// TwinCAT 3 PLC project PLC
// ProgramVersion: 3.1.4024.0
// libraries:
//   Tc2_Standard, * (Beckhoff Automation GmbH)
//   Tc2_System, * (Beckhoff Automation GmbH)
//   Tc3_Module, * (Beckhoff Automation GmbH)
// project tree:
//   DUTs/ DUT.TcDUT
//   / GlobalTextList.TcGTLO, PlcTask.TcTTO, Visualization Manager.TcVMO (not stored)
//   GVLs/ gHMI.TcGVL
//   POUs/FBs/ FB_Actuator.TcPOU, FB_StartingAlarm.TcPOU, FB_Contactor.TcPOU, FB_Debounce.TcPOU
//   POUs/Fs/ F_Scale.TcPOU
//   POUs/ MAIN.TcPOU, P_Control.TcPOU
//   VISUs/ VIS_Main.TcVIS
// real-time tasks:
//   TASK PlcTask: cycle T#10ms, priority 20, ADS port 350

CONFIGURATION PLC
    RESOURCE PLC ON TwinCAT3
        TASK PlcTask(INTERVAL := T#10ms, PRIORITY := 20);
        PROGRAM MAIN WITH PlcTask : MAIN;
    END_RESOURCE
END_CONFIGURATION

// ---- DUTs/DUT.TcDUT
TYPE DUT :
STRUCT
END_STRUCT
END_TYPE

// ---- GVLs/gHMI.TcGVL
{attribute 'qualified_only'}
VAR_GLOBAL
	Start: BOOL;
	Stop: BOOL;
	Reset: BOOL;
	Run: BOOL;
	Alarm: BOOL;
	Error: BOOL;	
END_VAR

// ---- POUs/MAIN.TcPOU
PROGRAM MAIN
VAR
END_VAR

P_Control();

END_PROGRAM

// ---- POUs/P_Control.TcPOU
PROGRAM P_Control
VAR
	fbStarter: FB_StartingAlarm;
	FB_Debounce_0: FB_Debounce;
	fbDebounce: FB_Debounce;
	fbContactor: FB_Contactor;
	simContactor: FB_Debounce;
END_VAR

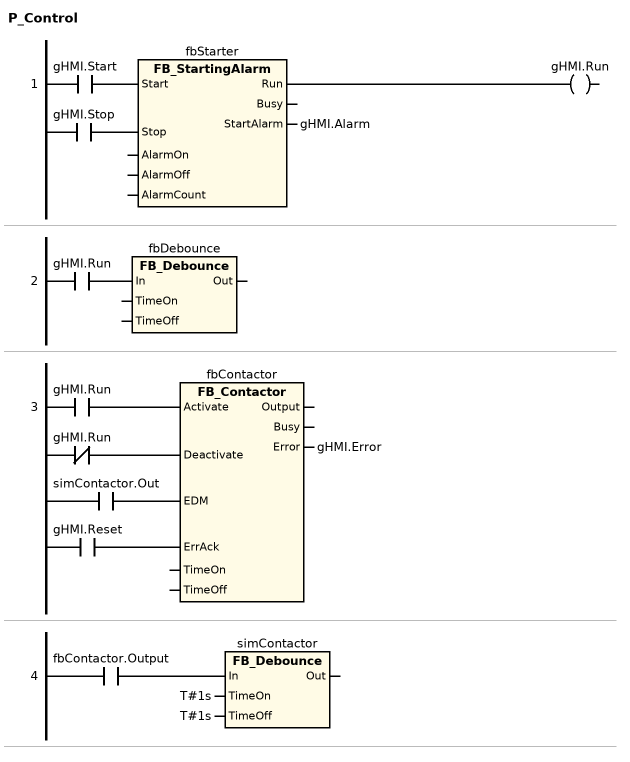
// NETWORK 1
fbStarter(Start := gHMI.Start, Stop := gHMI.Stop, StartAlarm => gHMI.Alarm); // FB_StartingAlarm
gHMI.Run := fbStarter.Run;

// NETWORK 2
fbDebounce(In := gHMI.Run); // FB_Debounce

// NETWORK 3
fbContactor(
    Activate := gHMI.Run,
    Deactivate := NOT gHMI.Run,
    EDM := simContactor.Out,
    ErrAck := gHMI.Reset,
    Error => gHMI.Error); // FB_Contactor

// NETWORK 4
simContactor(In := fbContactor.Output, TimeOn := T#1s, TimeOff := T#1s); // FB_Debounce

END_PROGRAM

// ---- POUs/FBs/FB_StartingAlarm.TcPOU
FUNCTION_BLOCK FB_StartingAlarm
VAR_INPUT
	Start: BOOL;
	Stop: BOOL;
	AlarmOn: TIME := T#500MS;
	AlarmOff: TIME := T#500MS;
	AlarmCount: UINT := 3;
END_VAR
VAR_OUTPUT
	Run: BOOL;
	Busy: BOOL;
	StartAlarm: BOOL;
END_VAR
VAR
	eState: (eInit, eIdle, eStarting, eRunning);
	eAlarmState: (eAlarmInit, eAlarmOn, eAlarmOff, eAlarmDone);
	rtrigStart: R_TRIG;
	rtrigStop: R_TRIG;
	tonAlarmOn: TON;
	tonAlarmOff: TON;
	nAlarmCount: UINT;
END_VAR

// Triggers
rtrigStop(CLK := Stop);

// Stop Interrrupt
IF rtrigStop.Q THEN
	eState := eInit;
END_IF

// State Machine
CASE eState OF
	eInit:
		Run := FALSE;
		Busy := FALSE;
		StartAlarm := FALSE;
		eAlarmState := eAlarmInit;	
		eState := eIdle;
		
	eIdle:
		IF Start THEN
			eState := eStarting;
		END_IF
		
	eStarting:
		Busy := TRUE;
		
		// Abort if Start not Held
		IF NOT Start THEN
			eState := eInit;
		END_IF
		
		// Alarm Sequence
		CASE eAlarmState OF
			eAlarmInit:
				tonAlarmOn.IN := FALSE;
				tonAlarmOn.PT := AlarmOn;
				tonAlarmOff.IN := FALSE;
				tonAlarmOff.PT := AlarmOff;
				nAlarmCount := 0;
				eAlarmState := eAlarmOn;
			eAlarmOn:
				tonAlarmOn.IN := TRUE;
				StartAlarm := TRUE;
				IF tonAlarmOn.Q THEN
					tonAlarmOn.IN := FALSE;
					eAlarmState := eAlarmOff;
				END_IF
			eAlarmOff:
				tonAlarmOff.IN := TRUE;
				StartAlarm := FALSE;
				IF tonAlarmOff.Q THEN
					tonAlarmOff.IN := FALSE;
					nAlarmCount := nAlarmCount + 1;
					IF nAlarmCount < AlarmCount THEN
						eAlarmState := eAlarmOn;
					ELSE
						eAlarmState := eAlarmDone;
					END_IF
				END_IF
				
			eAlarmDone:
				eState := eRunning;
		END_CASE
		
	eRunning:
		Busy := FALSE;
		Run := TRUE;	
END_CASE

// Call Function Blocks
tonAlarmOn();
tonAlarmOff();

END_FUNCTION_BLOCK

// ---- POUs/FBs/FB_Debounce.TcPOU
(* 	Disclaimer
	All sample code provided by Beckhoff Automation LLC are for illustrative purposes only and are provided “as is” and without any warranties, express or implied.
	Actual implementations in applications will vary significantly.
	Beckhoff Automation LLC shall have no liability for, and does not waive any rights in relation to, any code samples that it provides or the use of such code samples for any purpose.
*)
FUNCTION_BLOCK FB_Debounce
VAR_INPUT
	In: BOOL;
	TimeOn: TIME := T#2S;
	TimeOff: TIME := T#2S;
END_VAR
VAR_OUTPUT
	Out: BOOL;
END_VAR
VAR
	tonDelayOn: TON;
	tonDelayOff: TON;
END_VAR

// Set-Reset delay Timers
IF In THEN
	tonDelayOn.PT := TimeOn;
	tonDelayOn.IN := TRUE;
	tonDelayOff.IN := FALSE;
ELSE
	tonDelayOff.PT := TimeOff;
	tonDelayOff.IN := TRUE;
	tonDelayOn.IN := FALSE;
END_IF

// Set delayed Output
IF tonDelayOn.Q THEN
	Out := TRUE;
END_IF

// Reset delayed Output
IF tonDelayOff.Q THEN
	Out := FALSE;
END_IF

// Call function blocks
tonDelayOn();
tonDelayOff();

END_FUNCTION_BLOCK

// ---- POUs/FBs/FB_Contactor.TcPOU
(* 	Disclaimer
	All sample code provided by Beckhoff Automation LLC are for illustrative purposes only and are provided “as is” and without any warranties, express or implied.
	Actual implementations in applications will vary significantly.
	Beckhoff Automation LLC shall have no liability for, and does not waive any rights in relation to, any code samples that it provides or the use of such code samples for any purpose.
*)
FUNCTION_BLOCK FB_Contactor
VAR_INPUT
	Activate: BOOL;
	Deactivate: BOOL;
	EDM: BOOL;
	ErrAck: BOOL;
	TimeOn: TIME := T#3S;
	TimeOff: TIME := T#3S;
END_VAR
VAR_OUTPUT
	Output: BOOL;
	Busy: BOOL;
	Error: BOOL;
END_VAR
VAR
	eState :(eInit, eIdle, eActivate, eDeactivate, eError);
	tonWD: TON;
END_VAR

// Activating Watchdog
tonWD.IN := Output XOR EDM;
tonWD.PT := TimeOn;
IF tonWD.Q THEN
	Error := TRUE;
END_IF

// State Machine
CASE eState OF
	eInit:
		Output := FALSE;
		Busy := FALSE;
		Error := FALSE;
		eState := eIdle;
	
	eIdle:
		Busy := FALSE;
		IF Activate AND NOT Output THEN
			eState := eActivate;
		ELSIF NOT Activate AND Output THEN
			eState := eDeactivate;
		END_IF
		
	eActivate:
		Busy := TRUE;
		Output := TRUE;
		IF NOT Activate OR EDM THEN
			eState := eIdle;
		END_IF
	
	eDeactivate:
		Busy := TRUE;
		Output := FALSE;
		IF Activate OR NOT EDM THEN
			eState := eIdle;
		END_IF	
		
	eError:
		IF ErrAck THEN
			eState := eInit;
		END_IF
	
END_CASE

// Call function blocks
tonWD();

END_FUNCTION_BLOCK

// ---- POUs/FBs/FB_Actuator.TcPOU
(* 	Disclaimer
	All sample code provided by Beckhoff Automation LLC are for illustrative purposes only and are provided “as is” and without any warranties, express or implied.
	Actual implementations in applications will vary significantly.
	Beckhoff Automation LLC shall have no liability for, and does not waive any rights in relation to, any code samples that it provides or the use of such code samples for any purpose.
*)
FUNCTION_BLOCK FB_Actuator
VAR_INPUT
	Activate: BOOL;
	Deactivate: BOOL;
	EDM_Activated: BOOL;
	EDM_Deactivated: BOOL;
	ErrAck: BOOL;
	TimeOn: TIME := T#2S;
	TimeOff: TIME := T#2S;
END_VAR
VAR_OUTPUT
	Activated: BOOL;
	Busy: BOOL;
	Error: BOOL;
	ErrorId: UDINT;
END_VAR
VAR
	eState :(eInit, eIdle, eActivate, eDeactivate, eError);
	tonWD_On: TON;
	tonWD_Off: TON;
END_VAR

// Activating Watchdog
tonWD_On.IN := Activated AND NOT EDM_Activated;
tonWD_On.PT := TimeOn;
IF tonWD_On.Q THEN
	Error := TRUE;
	ErrorId := 1;
END_IF

// Deactivating Watchdog
tonWD_Off.IN := NOT Activated AND NOT EDM_Deactivated;
tonWD_Off.PT := TimeOff;
IF tonWD_Off.Q THEN
	Error := TRUE;
	ErrorId := 2;
END_IF

// State Machine
CASE eState OF
	eInit:
		Activated := FALSE;
		Busy := FALSE;
		Error := FALSE;
		ErrorId := 0;
		eState := eIdle;
	
	eIdle:
		Busy := FALSE;
		IF NOT Activated AND Activate THEN
			eState := eActivate;
		ELSIF Activated AND Deactivate THEN
			eState := eDeactivate;
		END_IF
		
	eActivate:
		Busy := TRUE;
		Activated := TRUE;
		IF NOT Activate OR EDM_Activated THEN
			eState := eIdle;
		END_IF
	
	eDeactivate:
		Busy := TRUE;
		Activated := FALSE;
		IF Activate OR EDM_Deactivated THEN
			eState := eIdle;
		END_IF	
		
	eError:
		IF ErrAck THEN
			eState := eInit;
		END_IF
	
END_CASE

// Call function blocks
tonWD_On();
tonWD_Off();

END_FUNCTION_BLOCK

// ---- POUs/Fs/F_Scale.TcPOU
(* 	Disclaimer
	All sample code provided by Beckhoff Automation LLC are for illustrative purposes only and are provided “as is” and without any warranties, express or implied.
	Actual implementations in applications will vary significantly.
	Beckhoff Automation LLC shall have no liability for, and does not waive any rights in relation to, any code samples that it provides or the use of such code samples for any purpose.
*)
FUNCTION F_Scale : LREAL
VAR_INPUT
	Value: INT;
END_VAR
VAR
END_VAR

// Percentage scale INT to LREAL 
F_Scale := Value/327.67;

// Limit to 0.0 - 100.0 percent
IF F_Scale < 0.0 THEN
	F_Scale := 0.0;
ELSIF F_Scale > 100.0 THEN
	F_Scale := 100.0;
END_IF

END_FUNCTION

// ---- VISUs/VIS_Main.TcVIS
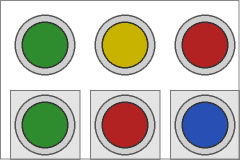
VISUALIZATION VIS_Main  // 240x160
    Lamp1 (10,10 70x70), variable: gHMI.Run, style: Lamp-Lamp1-Green
    Lamp1 (90,10 70x70), variable: gHMI.Alarm, style: Lamp-Lamp1-Yellow
    PushSwitch (10,90 70x70), variable: gHMI.Start, behaviour: TAP, style: Switch-PushSwitch-Green
    PushSwitch (90,90 70x70), variable: gHMI.Stop, behaviour: TAP, style: Switch-PushSwitch-Red
    PushSwitch (170,90 70x70), variable: gHMI.Reset, behaviour: TAP, style: Switch-PushSwitch-Blue
    Lamp1 (170,10 70x70), variable: gHMI.Error, style: Lamp-Lamp1-Red
END_VISUALIZATION
